FUNCTION_BLOCK ABSTRACT FB_StateMachine EXTENDS FB_Object IMPLEMENTS I_StateMachine
VAR_INPUT
END_VAR
VAR_OUTPUT
END_VAR
VAR
    _ipState:               I_State;
    _ipPrevState:           I_State;
    _nStateChangeCount:     UDINT := 0;
END_VAR

PROPERTY ipPrevState : I_State
GET
ipPrevState := THIS^._ipPrevState;
END_GET
END_PROPERTY

PROPERTY ipState : I_State
GET
ipState := THIS^._ipState;
END_GET
END_PROPERTY

METHOD SetState : BOOL
VAR_INPUT
    newState:           I_State;
END_VAR
IF THIS^.ipState <> newState THEN
    THIS^._ipState.OnExit();

    THIS^._ipPrevState := _ipState;
    THIS^._ipState := newState;

    THIS^._ipState.OnEntry();

    THIS^._nStateChangeCount := THIS^._nStateChangeCount + 1;

    SetState := TRUE;
END_IF
END_METHOD

END_FUNCTION_BLOCK

(* stored: Version 1.1.0.1, ProductVersion 3.1.4024.12
   POU FB_StateMachine: Id {fde30d05-33cb-4c8b-b55e-62aa88e8a800}, SpecialFunc None
   Property ipPrevState: Id {dd37e782-3259-48d5-bbdd-e492214b4e1d}
   Get Get: Id {e615f0e3-c5fd-4003-a6dc-12e9df41e5ea}
   Property ipState: Id {bc54c102-419f-4792-8ddb-88a43ac6e58c}
   Get Get: Id {e6c63ae4-e32d-4571-9341-0970144ab421}
   Method SetState: Id {c0a40504-cddb-40b7-affb-fd6284bdb099} *)
